FUNCTION_BLOCK Hour_Meter_FB
VAR_INPUT
	Running : BOOL;
END_VAR
VAR_OUTPUT
	Runtime_Hours : REAL;
END_VAR
VAR
	Running_Temp : BOOL;
	Minute_Timer : TON;
	Minutes : REAL;
	Hours : REAL;
	Elapsed : TIME;
END_VAR

Minute_Timer(IN:=Running_Temp , PT:=T#60S , Q=>, ET=>Elapsed );

IF Running THEN
	Running_Temp := TRUE;
END_IF
IF Minute_Timer.Q THEN
	Running_Temp := FALSE;
	Minutes := Minutes + 1;
END_IF
IF Minutes >= 60 THEN
	Minutes := 0;
	Hours := Hours + 1;
END_IF

Runtime_Hours := Hours;

END_FUNCTION_BLOCK

(* stored: Version 1.1.0.1, ProductVersion 3.1.4024.12
   POU Hour_Meter_FB: Id {fb40b7af-9bcc-47ec-87b2-16f4c6c8bd00}, SpecialFunc None *)
